ABB RAPID module: 0005D076

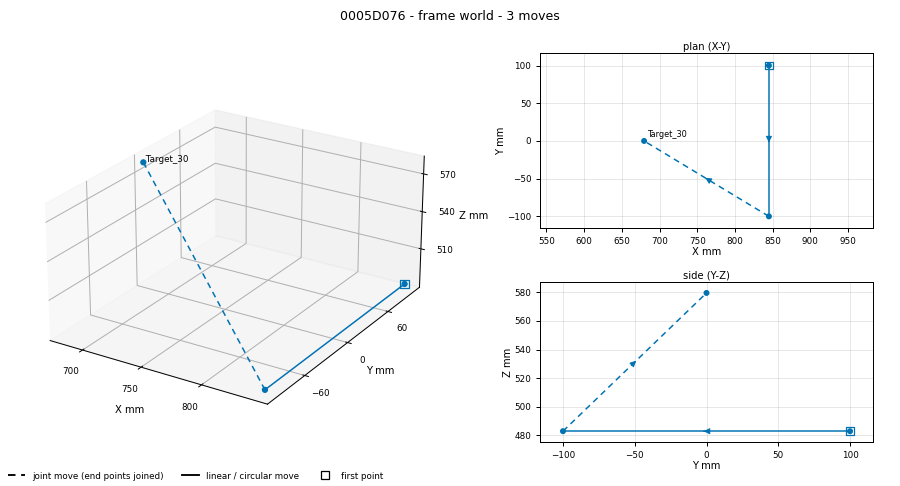
[picture p0: tool path of 0005D076 in frame world, 3 of 3 moves have a stored position in this frame; points joined in program order, loops and branches not executed]
MODULE Module1
    CONST robtarget Target_50:=[[506.291651246,0,679.5],[0.5,0,0.866025404,0],[0,0,0,0],[9E+09,9E+09,9E+09,9E+09,9E+09,9E+09]];
    CONST robtarget Target_30:=[[679.496731982,0,579.499999962],[0.5,0.5,0.5,0.5],[0,0,1,1],[9E+09,9E+09,9E+09,9E+09,9E+09,9E+09]];
    !***********************************************************
    !
    ! Module:  Module1
    !
    ! Description:
    !   <Insert description here>
    !
    ! Author: q
    !
    ! Version: 1.0
    !
    !***********************************************************


    !***********************************************************
    !
    ! Procedure main
    !
    !   This is the entry point of your program
    !
    !***********************************************************
    PROC Path_10()
        MoveJ [[845,100,483],[0.574751622,0.411898872,0.565053226,0.425105569],[0,0,-1,1],[9E+09,9E+09,9E+09,9E+09,9E+09,9E+09]],v500,fine,tool0\WObj:=wobj0;
        MoveL [[845,-100,483],[0.574751622,0.411898872,0.565053226,0.425105569],[-1,-1,1,1],[9E+09,9E+09,9E+09,9E+09,9E+09,9E+09]],vmax,fine,tool0\WObj:=wobj0;
        MoveJ Target_30,v500,z50,tool0\WObj:=wobj0;
    ENDPROC
ENDMODULE
